(* CODESYS project CAN_MIR3502.20200622.1.project
   Description: Receives some incoming messages and echoes them with CAN-ID +1
   Title: CAN Bus API Example
   Version: 1.0.0.0
   Company: 3S - Smart Software Solutions GmbH
   Author: 3S - Smart Software Solutions GmbH

Project tree, tasks and I/O mapping:
  Device : Changsha-Cyber-MI-linux, Changsha Cyber-MI Co., Ltd., version 3.5.10.40
    application Application
      libraries: CAN API, 1.0.0.3 (3S - Smart Software Solutions GmbH); Standard, * (System)
      task MainTask (cyclic, interval 10 ms, priority 16, watchdog 100 ms x 10) calls prg_mir3502
      function blocks/
        function block MsgProcessorMIR3502 [ST]: ProcessMessage
        function block FB_MIR3502_CAN [ST]: setup_sendmsg
        function block fb_avg [ST]
      global variables GVL
      program prg_mir3502 [ST]
      trace Trace (task MainTask): prg_mir3502.ai_00
    SoftMotion General Axis Pool
    IoDrvMIC7001 : IoDrvMIC7001, Cyber-MI, version 19.1.1
        unmapped channels: Ai00@C16, Ai01@C28, Ai02@C17, Ai03@C29, Ai04@C30, Ai05@C19, Ai06@C31, Ai07@C20, Ai08@C18, Ai09@D18, Ai10@D20, Ai11@D31, Ai12@D19, Ai13@D30, Ai14@D29, Ai15@D17, Ai16@D28, Ai17@D16, Ai18-Do00@C25, Ai19-Do01@C24, Ai20-Do02@C13, Ai21-Do03@C01, Ai22-Do04@C03, Ai23-Do05@C04, Ai24-Do06@C05, Ai25-Do07@C06, Ai26-Do08@C08, Ai27-Do09@C09, Ai28-Do10@C10, Ai29-Do11@C11, Ai30-Do12@D34, Ai31-Do13@D35, Ai32-Do14@D23, Ai33-Do15@D12, Ai34-Do16@D10, Ai35-Do17@D09, Ai36-Do18@D08, Ai37-Do19@D07, Ai38-Do20@D05, Ai39-Do21@D04,
          Ai40-Do22@D03, Ai41-Do23@D02, Ai42-Do24@C23, Ai43-Do25@C35, Ai44-Do26@D24, Ai45-Do27@D13, Ai46-Ao00@C22, Ai47-Ao01@D14, Ai48_Pi02, Ai49_Out5V, Ai50_VCC, Ai51_VCC_L, Ai52_VCC_R, Ai53_Pwm-i0, Ai54_Pwm-i1, Ai55_Pwm-i2, Ai56_Pwm-i3, Ai57_CPU-T, Ai58_G-x, Ai59_G-y, Ai60_G-z, Ai61-reserved, Ai62-IO-cntr, Ai63-CDS-cntr, Di00-Ai00@C16, Di01-Ai01@C28, Di02-Ai02@C17, Di03-Ai03@C29, Di04-Ai04@C30, Di05-Ai05@C19, Di06-Ai06@C31, Di07-Ai07@C20, Di08-Ai08@C18, Di09-Ai09@D18, Di10-Ai10@D20, Di11-Ai11@D31, Di12-Ai12@D19, Di13-Ai13@D30, Di14-Ai14@D29, Di15-Ai15@D17,
          Di16-Ai16@D28, Di17-Ai17@D16, Di18-Ai18@C25, Di19-Ai19@C24, Di20-Ai20@C13, Di21-Ai21@C01, Di22-Ai22@C03, Di23-Ai23@C04, Di24-Ai24@C05, Di25-Ai25@C06, Di26-Ai26@C08, Di27-Ai27@C09, Di28-Ai28@C10, Di29-Ai29@C11, Di30-Ai30@D34, Di31-Ai31@D35, Di32-Ai32@D23, Di33-Ai33@D12, Di34-Ai34@D10, Di35-Ai35@D09, Di36-Ai36@D08, Di37-Ai37@D07, Di38-Ai38@D05, Di39-Ai39@D04, Di40-Ai40@D03, Di41-Ai41@D02, Di42-Ai42@C23, Di43-Ai43@C35, Di44-Ai44@D24, Di45-Ai45@D13, Di46-Ai46@C22, Di47-Ai47@D14, Di48-Pi00@C15, Di49-Pi01@C14, Di50-Pi02@D22, Di51-Pi03@D21, Di52-reserved, Di53-reserved, Di54-reserved, Di55-reserved,
          Di56-reserved, Di57-reserved, Di58-reserved, Di59-reserved, Di60-reserved, Di61-reserved, Di62-reserved, Di63-reserved, Pi00-Di48@C15, Pi01-Di49@C14, Pi02-Di50@D22, Pi03-Di51@D21, Do00-Ai18@C25, Do01-Ai19@C24, Do02-Ai20@C13, Do03-Ai21@C01, Do04-Ai22@C03, Do05-Ai23@C04, Do06-Ai24@C05, Do07-Ai25@C06, Do08-Ai26@C08, Do09-Ai27@C09, Do10-Ai28@C10, Do11-Ai29@C11, Do12-Ai30@D34, Do13-Ai31@D35, Do14-Ai32@D23, Do15-Ai33@D12, Do16-Ai34@D10, Do17-Ai35@D09, Do18-Ai36@D08, Do19-Ai37@D07, Do20-Ai38@D05, Do21-Ai39@D04, Do22-Ai40@D03, Do23-Ai41@D02, Do24-Ai42@C23, Do25-Ai43@C35, Do26-Ai44@D24, Do27-Ai45@D13,
          Do28-Pwmi00@C33, Do29-Pwmi01@C34, Do30-Pwmi02@D25, Do31-Pwmi03@D26, PWM00@C25, PWM01@C24, PWM02@C13, PWM03@C01, PWM04@C03, PWM05@C04, PWM06@C05, PWM07@C06, PWM08@C08, PWM09@C09, PWM10@C10, PWM11@C11, PWM12@D34, PWM13@D35, PWM14@D23, PWM15@D12, PWM16@D10, PWM17@D09, PWM18@D08, PWM19@D07, PWM20@D05, PWM21@D04, PWM22@D03, PWM23@D02, PWM24@C23, PWM25@C35, PWM26@D24, PWM27@D13, PWM28-Pwmi00@C33, PWM29-Pwmi01@C34, PWM30-Pwmi02@D25, PWM31-Pwmi03@D26, PWM_I_0@C33, PWM_I_1@C34, PWM_I_2@D25, PWM_I_3@D26,
          Ao00-Ai46@C22, Ao01-Ai47@D14, LED_run, LED_err, LED_usr, ctrl_ai_raw, ctrl_adjust, ctrl_adj0, ctrl_adj1, ctrl_adj2, ctrl_adj3, disable_5V
*)

// Device/Application/GVL
VAR_GLOBAL

END_VAR

// Device/Application/prg_mir3502
PROGRAM prg_mir3502
VAR
	// CAN 0 ,  250K bps,  buffer size: 100
	CanConfig	: CAN.DRIVER_CONFIG := (usiNetwork:= 0, uiBaudrate:= 250, ctMessages:= 100);
	CANdriver	: CAN.CANBus_29bit :=  (DriverConfig:= CanConfig);
	
	// MIR3502
	MIR3502 : FB_MIR3502_CAN := (xEnable := TRUE);
	avg_ai00:fb_avg := (num := 32);
	
	ai_00_raw:DINT;
	ai_00 : DINT;
	ai_06 : DINT;
	ai_12 : DINT;
    ai_pwmi00 :DINT;
    ai_pwmi01 :DINT;
END_VAR


/// Run  the CAN Driver
CANdriver(DriverConfig:= CanConfig, eError=> );

MIR3502(CANdriver := CANdriver);

//设置扩展IO模块的DO， PWM
MIR3502.xDO[3] := TRUE;
//MIR3502.xDO[23] := TRUE;

//设置哪些AI需要读取，没有设置的AI值不会送到主控制器，以降低CAN总线负载率
MIR3502.xEnable_AI[00] := TRUE;
MIR3502.xEnable_AI[06] := TRUE;
MIR3502.xEnable_AI[12] := TRUE;
MIR3502.xEnable_AI[24] := TRUE;
MIR3502.xEnable_AI[28] := TRUE;


//读取扩展IO模块的AI
ai_00_raw := MIR3502.uiAI[0];
avg_ai00(in_val := ai_00_raw, out_val => ai_00);
ai_06 := MIR3502.uiAI[6];
ai_12 := MIR3502.uiAI[12];
ai_pwmi00 := MIR3502.uiAI[30];
ai_pwmi01 := MIR3502.uiAI[31];

END_PROGRAM

// Device/Application/function blocks/FB_MIR3502_CAN
FUNCTION_BLOCK FB_MIR3502_CAN
VAR_INPUT
	xEnable:BOOL := FALSE;
	xEnable_AI:ARRAY[0..31] OF BOOL := [32(FALSE)];
	xDO:ARRAY[0..23] OF BOOL := [24(FALSE)];
	uiPWM:ARRAY[0..1] OF UINT := [2(0)];
END_VAR
VAR_IN_OUT
	CANdriver	: CAN.CANBus_29bit;
END_VAR
VAR_OUTPUT
	uiAI:ARRAY[0..31] OF UINT;
    xDI:ARRAY[0..31] OF BOOL;
    Vcc:UINT;
    xError:BOOL := FALSE;
    sError:STRING(128) := 'No Error';	
	uiStat : UINT := 0;
END_VAR
VAR
	stat:UINT := 0;
	i :UINT := 0;
	recver:can.RECEIVER_AREA;
	areaReceiver:CAN.CANAreaReceiver;
	msgProcessor:MsgProcessorMIR3502;
	hAreaReceiver	: CAN.CAA.HANDLE := CAN.CAA.gc_hINVALID;
	bData:BYTE;
	msg_send :CAN.MESSAGE;
	msg_recv :CAN.MESSAGE;
END_VAR


CASE stat OF
0:
	FOR i := 0 TO 31 DO
		xEnable_AI[i] := FALSE;
		uiAI[i] := 0;
	END_FOR	
	
	FOR i := 0 TO 23 DO
		xDO[i] := FALSE;
		xDI[i] := FALSE;
	END_FOR
	
	FOR i := 0 TO 1 DO
		uiPWM[i] := 0;
	END_FOR
	
	Vcc := 0;
	xError := FALSE;
	sError := 'No Error';
	
	recver.dwIdStart := 300;
	recver.dwIdEnd := 308;
	recver.xRTRMask := FALSE;
	recver.xRTRValue := FALSE;
	recver.xTransmitMask := FALSE;
	recver.xTransmitValue := FALSE;

	hAreaReceiver := CANdriver.GetAreaReceiver(recver, eError=>);

	stat := 10;
	
10:  //wait enable
	IF xEnable THEN
		stat := 20;
	END_IF

20: //send
	setup_sendmsg();
	CANdriver.SendMessage(msg_send, eError=>);
	stat := 30;

30: //wait for receive
	stat := 20;  //send next msg
	
END_CASE

uiStat := stat;

CANdriver.ReceiveMessage(hReceiver := hAreaReceiver, itfMsgProcessor := msgProcessor, tTimeLimit := T#5MS, eError=>);

msgProcessor(CANdriver := CANdriver);

FOR i := 0 TO 31 DO
	uiAI[i] := msgProcessor.uiAI[i];
	xDI[i] := msgProcessor.xDI[i];
	Vcc := msgProcessor.Vcc;
END_FOR

ACTION setup_sendmsg:
	bData.0 := xDO[0]; 
	bData.1 := xDO[1];
	bData.2 := xDO[2];
	bData.3 := xDO[3];
	bData.4 := xDO[4];
	bData.5 := xDO[5];
	bData.6 := xDO[6];
	bData.7 := xDO[7];
	msg_send.abyData[0] := bData;
	
	bData.0 := xDO[8]; 
	bData.1 := xDO[9];
	bData.2 := xDO[10];
	bData.3 := xDO[11];
	bData.4 := xDO[12];
	bData.5 := xDO[13];
	bData.6 := xDO[14];
	bData.7 := xDO[15];
	msg_send.abyData[1] := bData;	
	
	bData.0 := xDO[16]; 
	bData.1 := xDO[17];
	bData.2 := xDO[18];
	bData.3 := xDO[19];
	bData.4 := xDO[20];
	bData.5 := xDO[21];
	bData.6 := xDO[22];
	bData.7 := xDO[23];
	msg_send.abyData[2] := bData;	

	bData.0 := NOT (xEnable_AI[0] OR xEnable_AI[1] OR xEnable_AI[2] OR xEnable_AI[3]) ; 
	bData.1 := NOT (xEnable_AI[4] OR xEnable_AI[5] OR xEnable_AI[6] OR xEnable_AI[7]) ; 
	bData.2 := NOT (xEnable_AI[8] OR xEnable_AI[9] OR xEnable_AI[10] OR xEnable_AI[11]) ; 
	bData.3 := NOT (xEnable_AI[12] OR xEnable_AI[13] OR xEnable_AI[14] OR xEnable_AI[15]) ; 
	bData.4 := NOT (xEnable_AI[16] OR xEnable_AI[17] OR xEnable_AI[18] OR xEnable_AI[19]) ; 
	bData.5 := NOT (xEnable_AI[20] OR xEnable_AI[21] OR xEnable_AI[22] OR xEnable_AI[23]) ; 
	bData.6 := NOT (xEnable_AI[24] OR xEnable_AI[25] OR xEnable_AI[26] OR xEnable_AI[27]) ; 
	bData.7 := NOT (xEnable_AI[28] OR xEnable_AI[29] OR xEnable_AI[30] OR xEnable_AI[31]) ; 
	msg_send.abyData[3] := bData;	
	
	bData := ANY_TO_BYTE(uiPWM[0] MOD 256);
	msg_send.abyData[4] := bData;
	
	bData := ANY_TO_BYTE(uiPWM[0] / 256);
	msg_send.abyData[5] := bData;
	
	bData := ANY_TO_BYTE(uiPWM[1] MOD 256);
	msg_send.abyData[6] := bData;
	
	bData := ANY_TO_BYTE(uiPWM[1] / 256);
	msg_send.abyData[7] := bData;
	
	msg_send.udiCanID := 400;
	msg_send.usiDataLength := 8;
	msg_send.xIs29BitMessage := FALSE;
	msg_send.xRTR := FALSE;
END_ACTION

END_FUNCTION_BLOCK

// Device/Application/function blocks/MsgProcessorMIR3502
FUNCTION_BLOCK MsgProcessorMIR3502 IMPLEMENTS CAN.IMessageProcessor
VAR_IN_OUT
	CANdriver	: CAN.CANBus_29bit;
END_VAR
VAR_OUTPUT
	uiAI:ARRAY[0..31] OF UINT;
    xDI:ARRAY[0..31] OF BOOL;
    Vcc:UINT;	
END_VAR
VAR
	_pCANdriver : POINTER TO CAN.CANBus_29bit;
END_VAR

_pCANdriver := ADR(CANdriver);

METHOD ProcessMessage
VAR_IN_OUT
	(* The messages received by the receiver *)
	Message	: CAN.RxMessage;
END_VAR

VAR
	id:UDINT;
END_VAR
IF _pCANdriver = 0 THEN
	RETURN;
END_IF

id := Message.udiCanID;

CASE id OF 
300:  //ai-00  ~  ai-03
	uiAI[0] := ANY_TO_UINT(Message.abyData[1])*256 + Message.abyData[0];
	uiAI[1] := ANY_TO_UINT(Message.abyData[3])*256 + Message.abyData[2];
	uiAI[2] := ANY_TO_UINT(Message.abyData[5])*256 + Message.abyData[4];
	uiAI[3] := ANY_TO_UINT(Message.abyData[7])*256 + Message.abyData[6];
 301:
	uiAI[4] := ANY_TO_UINT(Message.abyData[1])*256 + Message.abyData[0];
	uiAI[5] := ANY_TO_UINT(Message.abyData[3])*256 + Message.abyData[2];
	uiAI[6] := ANY_TO_UINT(Message.abyData[5])*256 + Message.abyData[4];
	uiAI[7] := ANY_TO_UINT(Message.abyData[7])*256 + Message.abyData[6];
 302:
	uiAI[8] := ANY_TO_UINT(Message.abyData[1])*256 + Message.abyData[0];
	uiAI[9] := ANY_TO_UINT(Message.abyData[3])*256 + Message.abyData[2];
	uiAI[10] := ANY_TO_UINT(Message.abyData[5])*256 + Message.abyData[4];
	uiAI[11] := ANY_TO_UINT(Message.abyData[7])*256 + Message.abyData[6];
 303:
	uiAI[12] := ANY_TO_UINT(Message.abyData[1])*256 + Message.abyData[0];
	uiAI[13] := ANY_TO_UINT(Message.abyData[3])*256 + Message.abyData[2];
	uiAI[14] := ANY_TO_UINT(Message.abyData[5])*256 + Message.abyData[4];
	uiAI[15] := ANY_TO_UINT(Message.abyData[7])*256 + Message.abyData[6];
 304:
	uiAI[16] := ANY_TO_UINT(Message.abyData[1])*256 + Message.abyData[0];
	uiAI[17] := ANY_TO_UINT(Message.abyData[3])*256 + Message.abyData[2];
	uiAI[18] := ANY_TO_UINT(Message.abyData[5])*256 + Message.abyData[4];
	uiAI[19] := ANY_TO_UINT(Message.abyData[7])*256 + Message.abyData[6];
 305:
	uiAI[20] := ANY_TO_UINT(Message.abyData[1])*256 + Message.abyData[0];
	uiAI[21] := ANY_TO_UINT(Message.abyData[3])*256 + Message.abyData[2];
	uiAI[22] := ANY_TO_UINT(Message.abyData[5])*256 + Message.abyData[4];
	uiAI[23] := ANY_TO_UINT(Message.abyData[7])*256 + Message.abyData[6];
 306:
	uiAI[24] := ANY_TO_UINT(Message.abyData[1])*256 + Message.abyData[0];
	uiAI[25] := ANY_TO_UINT(Message.abyData[3])*256 + Message.abyData[2];
	uiAI[26] := ANY_TO_UINT(Message.abyData[5])*256 + Message.abyData[4];
	uiAI[27] := ANY_TO_UINT(Message.abyData[7])*256 + Message.abyData[6];
 307:
	uiAI[28] := ANY_TO_UINT(Message.abyData[1])*256 + Message.abyData[0];
	uiAI[29] := ANY_TO_UINT(Message.abyData[3])*256 + Message.abyData[2];
	uiAI[30] := ANY_TO_UINT(Message.abyData[5])*256 + Message.abyData[4];
	uiAI[31] := ANY_TO_UINT(Message.abyData[7])*256 + Message.abyData[6];
 308:  //DI00 ~ DI23   and  Vcc
	xDi[0] :=  Message.abyData[0].0;
	xDi[1] :=  Message.abyData[0].1;
	xDi[2] :=  Message.abyData[0].2;
	xDi[3] :=  Message.abyData[0].3;
	xDi[4] :=  Message.abyData[0].4;
	xDi[5] :=  Message.abyData[0].5;
	xDi[6] :=  Message.abyData[0].6;
	xDi[7] :=  Message.abyData[0].7;
	
	xDi[8] :=  Message.abyData[1].0;
	xDi[9] :=  Message.abyData[1].1;
	xDi[10] :=  Message.abyData[1].2;
	xDi[11] :=  Message.abyData[1].3;
	xDi[12] :=  Message.abyData[1].4;
	xDi[13] :=  Message.abyData[1].5;
	xDi[14] :=  Message.abyData[1].6;
	xDi[15] :=  Message.abyData[1].7;

	xDi[16] :=  Message.abyData[2].0;
	xDi[17] :=  Message.abyData[2].1;
	xDi[18] :=  Message.abyData[2].2;
	xDi[19] :=  Message.abyData[2].3;
	xDi[20] :=  Message.abyData[2].4;
	xDi[21] :=  Message.abyData[2].5;
	xDi[22] :=  Message.abyData[2].6;
	xDi[23] :=  Message.abyData[2].7;

	xDi[24] :=  Message.abyData[3].0;
	xDi[25] :=  Message.abyData[3].1;
	xDi[26] :=  Message.abyData[3].2;
	xDi[27] :=  Message.abyData[3].3;
	xDi[28] :=  Message.abyData[3].4;
	xDi[29] :=  Message.abyData[3].5;
	xDi[30] :=  Message.abyData[3].6;
	xDi[31] :=  Message.abyData[3].7;	
	
	Vcc := ANY_TO_UINT(Message.abyData[7])*256 + Message.abyData[6];
END_CASE
END_METHOD

END_FUNCTION_BLOCK

// Device/Application/function blocks/fb_avg
FUNCTION_BLOCK fb_avg
VAR_INPUT
	in_val:DINT;
	num:DINT := 10;
END_VAR
VAR_OUTPUT
	out_val:DINT;
END_VAR
VAR
	num_max : DINT := 255;
	data:ARRAY[1..255] OF DINT; //需要与上面的num_max保持一致
	ptr :UINT := 1;
	i: DINT;
	sum: DINT;
END_VAR

IF num <1 THEN
	out_val := 0;
	RETURN;
END_IF
IF num > num_max THEN
	num := num_max;
END_IF

data[ptr] := in_val;
ptr := ptr + 1;
IF ptr > num THEN
	ptr := 1;
END_IF

sum := 0;
FOR i := 1 TO num DO
	sum := sum + data[i];
END_FOR

out_val := sum/num;

END_FUNCTION_BLOCK
